FUNCTION_BLOCK PVPROG_LOCK (* Blocks output events and input data for FB_PVPROG *)
  (* Standard: 61499; Classification: Event Processing; Description: Blocks output events and input data for FB_PVPROG after receival of L event until arrival of UL event. In the unlocked state (after receiving U event), the L input event is passed to the LO output event and the input data is passed to the output data. Receiving an L input event puts the FB into a locked state, in which L events and their respective data are not forwarded. The FB can be moved from a locked state into an unlocked state with a U event input, which also generates a UO event output. *)
  (* Version 1.0, 2017-05-22, Marc Jakobi, HTW Berlin *)
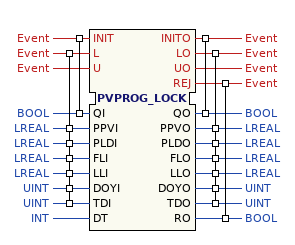
  EVENT_INPUT
    INIT WITH QI; (* Initialization Event *)
    L WITH PPVI, PLDI, FLI, LLI, DOYI, TDI; (* Lock Event *)
    U; (* Unlock Event *)
  END_EVENT
  EVENT_OUTPUT
    INITO WITH QO; (* Initialization Output Event *)
    LO WITH PPVO, PLDO, FLO, LLO, DOYO, TDO; (* Lock Confirmation *)
    UO; (* Unlock Confirmation *)
    REJ WITH RO; (* Rejected Request Notification *)
  END_EVENT
  VAR_INPUT
    QI : BOOL; (* Input event qualifier *)
    PPVI : LREAL; (* PV power in W *)
    PLDI : LREAL; (* Load in W *)
    FLI : LREAL; (* Feed-in limitation in W (0 for none) *)
    LLI : LREAL; (* Load limit in W (0 for none) *)
    DOYI : UINT; (* Day of the year [1..365] *)
    TDI : UINT; (* Time of day [min] [0..1439] *)
    DT : INT; (* Frequency [min] at which to let data through *)
  END_VAR
  VAR_OUTPUT
    QO : BOOL; (* Output event qualifier *)
    PPVO : LREAL; (* PV power in W *)
    PLDO : LREAL; (* Load in W *)
    FLO : LREAL; (* Feed-in limitation in W (0 for none) *)
    LLO : LREAL; (* Load limit in W (0 for none) *)
    DOYO : UINT; (* Day of the year [1..365] *)
    TDO : UINT; (* Time of day [min] [0..1439] *)
    RO : BOOL; (* Rejection reason indicator. TRUE: Not enough time passed; FALSE: Currently locked *)
  END_VAR
  VAR
    TIMESINCELASTREQ : INT := -1; (* Time [min] between last update and current one *)
    LASTTIMESTEP : INT := -1; (* Time at the point of the last call of the prepareForecast algorithm *)
  END_VAR
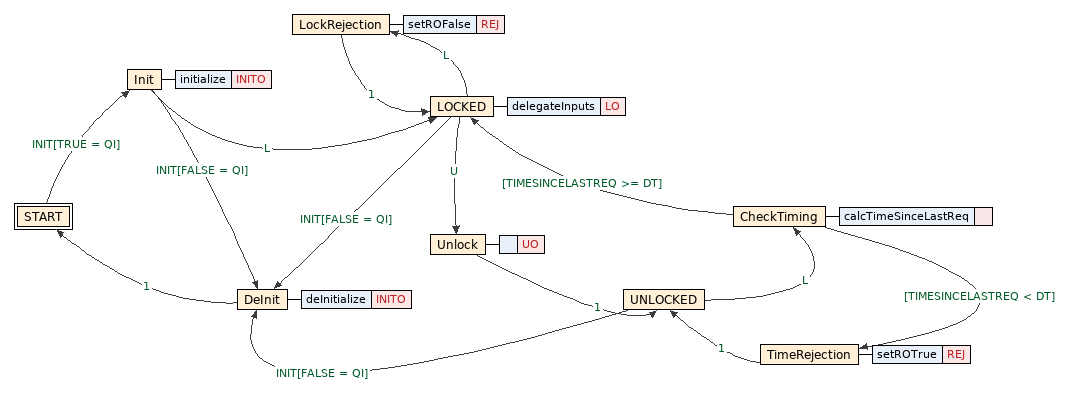
  EC_STATES
    START; (* Set Q and issue EO *)
    LOCKED : delegateInputs -> LO; (* Reset Q and issue EO *)
    UNLOCKED;
    Init : initialize -> INITO;
    DeInit : deInitialize -> INITO;
    CheckTiming : calcTimeSinceLastReq;
    Unlock : -> UO;
    TimeRejection : setROTrue -> REJ;
    LockRejection : setROFalse -> REJ;
  END_STATES
  EC_TRANSITIONS
    START TO Init := INIT[TRUE = QI];
    Init TO LOCKED := L;
    LOCKED TO DeInit := INIT[FALSE = QI];
    UNLOCKED TO DeInit := INIT[FALSE = QI];
    DeInit TO START := 1;
    Init TO DeInit := INIT[FALSE = QI];
    UNLOCKED TO CheckTiming := L;
    CheckTiming TO LOCKED := [TIMESINCELASTREQ >= DT];
    LOCKED TO Unlock := U;
    Unlock TO UNLOCKED := 1;
    CheckTiming TO TimeRejection := [TIMESINCELASTREQ < DT];
    TimeRejection TO UNLOCKED := 1;
    LOCKED TO LockRejection := L;
    LockRejection TO LOCKED := 1;
  END_TRANSITIONS
  ALGORITHM delegateInputs IN ST: (* delegates input variables to output variables *)
PPVO := PPVI;
PLDO := PLDI;
FLO := FLI;
LLO := LLI;
DOYO := DOYI;
TDO := TDI;
LASTTIMESTEP := TDI;
  END_ALGORITHM
  ALGORITHM initialize IN ST: (* initialization algorithm *)
LASTTIMESTEP := -1;
QO := TRUE;
  END_ALGORITHM
  ALGORITHM deInitialize IN ST: (* deinitialization algorithm *)
QO := FALSE;
  END_ALGORITHM
  ALGORITHM calcTimeSinceLastReq IN ST: (* calculates the time in minutes between the current and last requests *)
TIMESINCELASTREQ := UINT_TO_INT(TDI) - LASTTIMESTEP;
IF TIMESINCELASTREQ < 0 THEN // New day
	TIMESINCELASTREQ := DT;
END_IF;
  END_ALGORITHM
  ALGORITHM setROFalse IN ST: (* sets output RO to FALSE *)
RO := FALSE;
  END_ALGORITHM
  ALGORITHM setROTrue IN ST: (* sets output RO to TRUE *)
RO := TRUE;
  END_ALGORITHM
END_FUNCTION_BLOCK
